// Mitsubishi GX Works2 project: e04   PLC: Q02/Q02H

PROGRAM MAIN
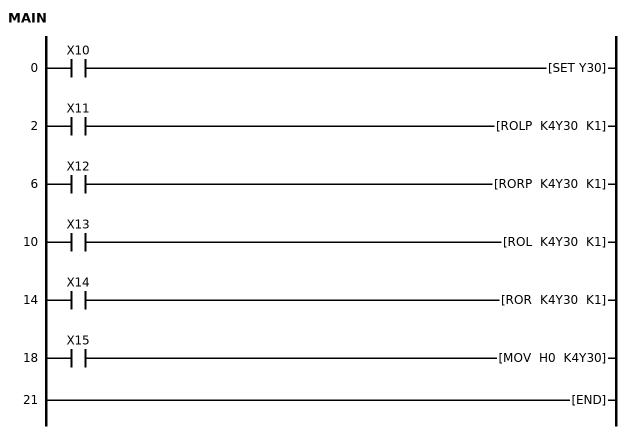
0     LD      X10
      SET     Y30
2     LD      X11
      ROLP    K4Y30 K1
6     LD      X12
      RORP    K4Y30 K1
10    LD      X13
      ROL     K4Y30 K1
14    LD      X14
      ROR     K4Y30 K1
18    LD      X15
      MOV     H0 K4Y30
21    END
END_PROGRAM
